INTERFACE I_XTS_Station EXTENDS I_CH_Object

METHOD AddMoverToQueue : HRESULT
VAR_INPUT
	ipMover : I_XTS_Mover;
END_VAR
END_METHOD

//Call this Methode whith seq 0->99, and wait each step until S_OK is returned
METHOD Configure : HRESULT
VAR_INPUT
	nSeq : UINT; //0->100
END_VAR
END_METHOD

{attribute 'monitoring':='call'}
PROPERTY CtsEmptySpaceInQueue : UDINT
GET
END_GET
END_PROPERTY

{attribute 'monitoring':='call'}
PROPERTY CtsMoversInQueue : UDINT
GET
END_GET
END_PROPERTY

METHOD DeleteMoversQueue : HRESULT
VAR_INPUT
END_VAR
END_METHOD

{attribute 'monitoring':='call'}
PROPERTY HR : HRESULT
GET
END_GET
END_PROPERTY

{attribute 'monitoring':='call'}
PROPERTY LUID : STRING
GET
END_GET
END_PROPERTY

{attribute 'monitoring':='call'}
PROPERTY MoverGapAtExit : LREAL
GET
END_GET
SET
END_SET
END_PROPERTY

{attribute 'monitoring':='call'}
PROPERTY MoverQueueSize : UINT
GET
END_GET
SET
END_SET
END_PROPERTY

{attribute 'monitoring':='call'}
PROPERTY MoversInPlace : BOOL
GET
END_GET
END_PROPERTY

{attribute 'monitoring':='call'}
PROPERTY MoversInQueue : REFERENCE TO ARRAY [0..(XtsParameterlist.MAX_MOVER_PER_SYSTEM-1)] OF I_XTS_Mover_PLC // Return a sorted list of movers in this zone. Index 0 is the mover in Front.
GET
END_GET
END_PROPERTY

{attribute 'monitoring':='call'}
PROPERTY MoverVelocityAtExit : LREAL
GET
END_GET
SET
END_SET
END_PROPERTY

{attribute 'monitoring':='call'}
PROPERTY PositionOnTrack : LREAL
GET
END_GET
END_PROPERTY

{attribute 'monitoring':='call'}
PROPERTY ReadyToRecvMovers : BOOL
GET
END_GET
SET
END_SET
END_PROPERTY

METHOD SendMoversToStation : HRESULT
VAR_INPUT
	sTargedStation : STRING;
END_VAR
END_METHOD

{attribute 'monitoring':='call'}
PROPERTY StationsAhead : I_XTS_Station
GET
END_GET
END_PROPERTY

END_INTERFACE

(* stored: Version 1.1.0.1, ProductVersion 3.1.4024.12
   Itf I_XTS_Station: Id {93173e7e-5f1f-41b7-9cae-ddf1ef2d2fc7}
   Method AddMoverToQueue: Id {dcf69248-1849-4ab5-a6f1-55dec9788659}
   Method Configure: Id {dfd1febc-b72b-4834-bea4-0048c8f97b04}
   Property CtsEmptySpaceInQueue: Id {80790399-3f9b-44a8-a885-28b318172fd5}
   Get Get: Id {500818d1-9da7-4f36-b8c4-0e920895a712}
   Property CtsMoversInQueue: Id {a57bef8b-97f7-4467-a0b2-f4bc8c7a4402}
   Get Get: Id {0accd52b-0b99-412b-8aee-2ae586f624e7}
   Method DeleteMoversQueue: Id {fb8db26b-4ead-4719-9871-bcdd0b308cc0}
   Property HR: Id {50cb5acf-1f27-4e58-a36a-fc1ef0412020}
   Get Get: Id {41afba73-6745-4f8e-8c07-ebb6ee366ce5}
   Property LUID: Id {80fdfa3d-95e5-40af-8b8a-1b721c812ed5}
   Get Get: Id {960fc52e-c825-46d7-9f7f-0336d3dd7aaa}
   Property MoverGapAtExit: Id {5cec660b-2c1a-4fe0-a842-d599f159e3f3}
   Get Get: Id {6e024805-9a5a-4187-af3a-31675f1cfed6}
   Set Set: Id {9225ed17-d2a6-41ac-a388-48da6877d1a0}
   Property MoverQueueSize: Id {d07e5abb-653c-4489-a199-5c48ad380e2d}
   Get Get: Id {c7ac416b-4571-4290-84b8-b24fb62928bb}
   Set Set: Id {ae6153c6-30f1-43d2-8eeb-56ab8c5b1c35}
   Property MoversInPlace: Id {6c2732a7-171c-473e-9dce-c93b33167f6b}
   Get Get: Id {37404813-753d-4c2e-a168-46ee3e8d956c}
   Property MoversInQueue: Id {72fa1f99-2d88-4fc8-a44a-15ceaadbab8d}
   Get Get: Id {46d8e947-1385-4541-8d64-3eb9f848c3ad}
   Property MoverVelocityAtExit: Id {7c8fef6f-8178-46e1-a440-896b17c90f80}
   Get Get: Id {84e145b2-a750-4419-a9f7-02fc13104142}
   Set Set: Id {0710baff-db39-417b-8e73-521eed5928a6}
   Property PositionOnTrack: Id {7d2c12fd-5cf9-479d-8ca9-098e54ea4d0a}
   Get Get: Id {56524df3-6b32-453e-ac1d-5e37753457a8}
   Property ReadyToRecvMovers: Id {caa39dfc-e0be-4923-986b-1578eaeb490b}
   Get Get: Id {0f055eb7-1aae-4886-8313-b660b15254bf}
   Set Set: Id {a74586e8-2c40-4339-9547-908e8aa7bc71}
   Method SendMoversToStation: Id {beedf22c-a16b-4887-8f1e-7ebc05099ac2}
   Property StationsAhead: Id {e35d3ecc-e3ff-4c39-a35b-bf61781b13ea}
   Get Get: Id {4442a0a4-c536-4116-bceb-a54a7d579086} *)
